FUNCTION_BLOCK AnalogInputParametersFB
VAR_INPUT
END_VAR
VAR_OUTPUT
	F_BT1: LREAL; // Frånluftstemperatur $(unit "°C")  
    T_BT2: LREAL; // Uteluftstemperatur $(unit "°C")
    T_BT3: LREAL; // Tilluftstemperatur (innan efterbehandling) $(unit "°C")
    H_BT1: LREAL; // Frysskyddstemperatur (används bara om värmebatteri (av vätsketyp) är installerat) $(unit "°C")
    T_BT1: LREAL; // Tilluftstemperatur (efter efterbehandling) $(unit "°C") 
    BT1: LREAL; // Utomhustemperatur (extern utegivare, T.BT2 används som utegivare som standard) $(unit "°C")
    BT2: LREAL; // Rumstemperatur (lokalgivare, används inte i bostadsaggregat) $(unit "°C")
    F_BT2: LREAL; // Avluftstemperatur (tillval) $(unit "°C")
	
    F_BP1: LREAL; // Tryckgivare Frånluftskanal $(unit "Pa")
    T_BP1: LREAL; // Tryckgivare Tilluftskanal $(unit "Pa")
    F_BP2: LREAL; // Tryckgivare Frånluftsfilter $(unit "Pa")
    T_BP2: LREAL; //  Tryckgivare uteluftsfilter $(unit "Pa")
    F_BP3: LREAL; // Tryckgivare VVX $(unit "Pa")
    T_BF1: LREAL; // Flödesgivare Tilluftsfläkt $(unit "m³/h")
    F_BF1: LREAL; // Flödesgivare Frånluftsfläkt $(unit "m³/h")	

	F_BT1_Error: BOOL; 
    T_BT2_Error: BOOL;
    T_BT3_Error: BOOL;
    H_BT1_Error: BOOL;
    T_BT1_Error: BOOL; 
    BT1_Error: BOOL;
    BT2_Error: BOOL;
    F_BT2_Error: BOOL;
	
    F_BP1_Error: BOOL;
    T_BP1_Error: BOOL;
    F_BP2_Error: BOOL;
    T_BP2_Error: BOOL;
    F_BP3_Error: BOOL;
    T_BF1_Error: BOOL;
    F_BF1_Error: BOOL;	

	F_BT1_EN: BOOL := TRUE; 
    T_BT2_EN: BOOL := TRUE;
    T_BT3_EN: BOOL := TRUE;
    H_BT1_EN: BOOL := FALSE;
    T_BT1_EN: BOOL := TRUE; 
    BT1_EN: BOOL := FALSE;
    BT2_EN: BOOL := FALSE;
    F_BT2_EN: BOOL := TRUE;
	
    F_BP1_EN: BOOL := TRUE;
    T_BP1_EN: BOOL := TRUE;
    F_BP2_EN: BOOL := TRUE;
    T_BP2_EN: BOOL := TRUE;
    F_BP3_EN: BOOL := TRUE;
    T_BF1_EN: BOOL := TRUE;
    F_BF1_EN: BOOL := TRUE;	
END_VAR
VAR
END_VAR

METHOD Update : BOOL
VAR_INPUT
	AI: REFERENCE TO GreenMasterAI_Base;
	AI2: REFERENCE TO GreenMasterAIU_Base;
	Parameters: REFERENCE TO GreenMasterBaseParameters;
END_VAR
IF NOT Parameters.System.Operation.Simulation THEN
	F_BT1 := AI.F_BT1;
	F_BT1_Error := AI.F_BT1_Error AND F_BT1_EN;
	T_BT2 := AI.T_BT2;
	T_BT2_Error := AI.T_BT2_Error AND T_BT2_EN;
	T_BT3 := AI.T_BT3;
	T_BT3_Error := AI.T_BT3_Error AND T_BT3_EN;
	H_BT1 := AI.H_BT1;
	H_BT1_Error := AI.H_BT1_Error AND H_BT1_EN;
	T_BT1 := AI.T_BT1; 
	T_BT1_Error := AI.T_BT1_Error AND T_BT1_EN;
	BT1 := AI.BT1;
	BT1_Error := AI.BT1_Error AND BT1_EN;
	BT2 := AI.BT2;
	BT2_Error := AI.BT2_Error AND BT2_EN;
	F_BT2 := AI.F_BT2;
	F_BT2_Error := AI.F_BT2_Error AND F_BT2_EN;
	F_BP1 := AI2.F_BP1;
	F_BP1_Error := AI2.F_BP1_Error AND F_BP1_EN;
	T_BP1 := AI2.T_BP1;
	T_BP1_Error := AI2.T_BP1_Error AND T_BP1_EN;
	F_BP2 := AI2.F_BP2;
	F_BP2_Error := AI2.F_BP2_Error AND F_BP2_EN;
	T_BP2 := AI2.T_BP2;
	T_BP2_Error := AI2.T_BP2_Error AND T_BP2_EN;
	F_BP3 := AI2.F_BP3;
	F_BP3_Error := AI2.F_BP3_Error AND F_BP3_EN;
	T_BF1 := AI2.T_BF1;
	T_BF1_Error := AI2.T_BF1_Error AND T_BF1_EN;
	F_BF1 := AI2.F_BF1;	
	F_BF1_Error := AI2.F_BF1_Error AND F_BF1_EN;
ELSE
	F_BT1_Error := FALSE;
	T_BT2_Error := FALSE;
	T_BT3_Error := FALSE;
	H_BT1_Error := FALSE;
	T_BT1_Error := FALSE;
	BT1_Error := FALSE;
	BT2_Error := FALSE;
	F_BT2_Error := FALSE;
	F_BP1_Error := FALSE;
	T_BP1_Error := FALSE;
	F_BP2_Error := FALSE;
	T_BP2_Error := FALSE;
	F_BP3_Error := FALSE;
	T_BF1_Error := FALSE;
	F_BF1_Error := FALSE;
END_IF
END_METHOD

END_FUNCTION_BLOCK

(* stored: Version 1.1.0.1, ProductVersion 3.1.4024.6
   POU AnalogInputParametersFB: Id {e766f1f7-f183-44ee-8a02-b37c486db9e7}, SpecialFunc None
   Method Update: Id {8483c25b-6617-4e28-ac3f-e8aa1724067f} *)
